FUNCTION_BLOCK Drum (* Composite Function Block Type *)
  (* Standard: 61499-2 *)
  (* Version 0.0, 2011-12-09, 4DIAC-IDE, 4DIAC-Consortium *)
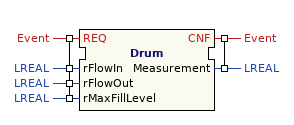
  EVENT_INPUT
    REQ WITH rFlowIn, rFlowOut, rMaxFillLevel; (* Normal Execution Request *)
  END_EVENT
  EVENT_OUTPUT
    CNF WITH Measurement; (* Execution Confirmation *)
  END_EVENT
  VAR_INPUT
    rFlowIn : LREAL; (* Input flow *)
    rFlowOut : LREAL; (* Output flow *)
    rMaxFillLevel : LREAL; (* Maximum fill level *)
  END_VAR
  VAR_OUTPUT
    Measurement : LREAL; (* Actual fill level *)
  END_VAR
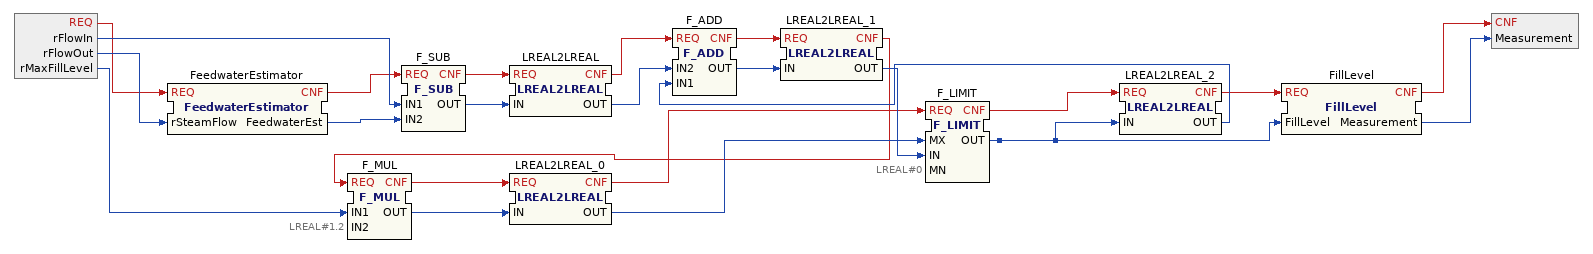
  FBS
    FeedwaterEstimator : FeedwaterEstimator;
    FillLevel : FillLevel;
    F_LIMIT : F_LIMIT(MN := LREAL#0);
    F_SUB : F_SUB;
    LREAL2LREAL : LREAL2LREAL;
    F_MUL : F_MUL(IN2 := LREAL#1.2);
    LREAL2LREAL_0 : LREAL2LREAL;
    F_ADD : F_ADD;
    LREAL2LREAL_1 : LREAL2LREAL;
    LREAL2LREAL_2 : LREAL2LREAL;
  END_FBS
  EVENT_CONNECTIONS
    REQ TO FeedwaterEstimator.REQ;
    FillLevel.CNF TO CNF;
    F_SUB.CNF TO LREAL2LREAL.REQ;
    F_MUL.CNF TO LREAL2LREAL_0.REQ;
    FeedwaterEstimator.CNF TO F_SUB.REQ;
    LREAL2LREAL.CNF TO F_ADD.REQ;
    LREAL2LREAL_0.CNF TO F_LIMIT.REQ;
    F_ADD.CNF TO LREAL2LREAL_1.REQ;
    LREAL2LREAL_1.CNF TO F_MUL.REQ;
    F_LIMIT.CNF TO LREAL2LREAL_2.REQ;
    LREAL2LREAL_2.CNF TO FillLevel.REQ;
  END_CONNECTIONS
  DATA_CONNECTIONS
    rFlowOut TO FeedwaterEstimator.rSteamFlow;
    FillLevel.Measurement TO Measurement;
    F_SUB.OUT TO LREAL2LREAL.IN;
    LREAL2LREAL_0.OUT TO F_LIMIT.MX;
    F_MUL.OUT TO LREAL2LREAL_0.IN;
    rMaxFillLevel TO F_MUL.IN1;
    rFlowIn TO F_SUB.IN1;
    FeedwaterEstimator.FeedwaterEst TO F_SUB.IN2;
    LREAL2LREAL.OUT TO F_ADD.IN2;
    F_LIMIT.OUT TO FillLevel.FillLevel;
    F_ADD.OUT TO LREAL2LREAL_1.IN;
    LREAL2LREAL_1.OUT TO F_LIMIT.IN;
    F_LIMIT.OUT TO LREAL2LREAL_2.IN;
    LREAL2LREAL_2.OUT TO F_ADD.IN1;
  END_CONNECTIONS
END_FUNCTION_BLOCK
